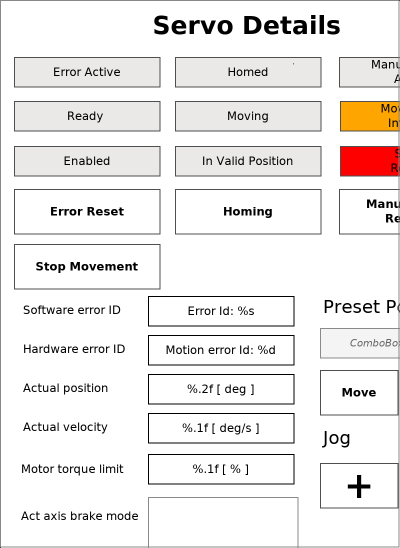
VISUALIZATION vAxisDetail  // 400x548
VAR_IN_OUT
	fbAxis: fb_ServoAxis;
	fbTableControl :FB_TableControl;
END_VAR
    Rectangle (0,0 495x856)
    Rectangle (339,189 146x45), "Manual mode Request", colour toggle: fbAxis.stHMI.bManualModeRequest
        toggle fbAxis.stHMI.bManualModeRequest
    Label (20,376 130x24), "Actual position"
    Label (20,415 130x24), "Actual velocity"
    Label (18,457 145x24), "Motor torque limit"
    Label (20,298 130x24), "Software error ID"
    Label (20,337 130x24), "Hardware error ID"
    Label (18,504 130x24), "Act axis brake mode"
    Label (18,544 130x24), "New brake mode"
    Frame (148,497 150x130)
        shows vAxisBrakeControl(fbData := MAIN.fbTableAxis)
    Rectangle (320,463 78x45), "+", colour toggle: fbAxis.stHMI.bJogForwardButton, input disabled if: fbAxis.iWorkStep_Axis<>15
        OnMouseDown: execute { fbAxis.stHMI.bJogForwardButton:=TRUE; }
        OnMouseLeave: execute { fbAxis.stHMI.bJogForwardButton :=FALSE; }
        OnMouseUp: execute { fbAxis.stHMI.bJogForwardButton :=FALSE; }
    Rectangle (405,463 74x45), "-", colour toggle: fbAxis.stHMI.bJogBackwardButton, input disabled if: fbAxis.iWorkStep_Axis<>15
        OnMouseDown: execute { fbAxis.stHMI.bJogBackwardButton:=TRUE; }
        OnMouseLeave: execute { fbAxis.stHMI.bJogBackwardButton:=FALSE; }
        OnMouseUp: execute { fbAxis.stHMI.bJogBackwardButton:=FALSE; }
    Label (149,8 196x34), "Servo Details"
    ComboBoxInteger (320,328 150x30), variable: fbAxis.stHMI.iManualPositionSelected, input disabled if: fbAxis.iWorkStep_Axis<>15
    Rectangle (320,370 78x45), "Move", colour toggle: fbAxis.stHMI.bGoToSelectedPosition, input disabled if: fbAxis.iWorkStep_Axis<>15
        OnMouseDown: execute { fbAxis.stHMI.bGoToSelectedPosition:=TRUE; }
        OnMouseLeave: execute { fbAxis.stHMI.bGoToSelectedPosition:=FALSE; }
        OnMouseUp: execute { fbAxis.stHMI.bGoToSelectedPosition:=FALSE; }
    Label (320,423 161x30), "Jog"
    Label (320,292 161x30), "Preset Position"
    Rectangle (175,189 146x45), "Homing", colour toggle: fbAxis.iWorkStep_Axis =20 OR fbAxis.iWorkStep_Axis =21
        OnMouseDown: execute { fbAxis.mFullHoming(); }
    Rectangle (339,57 146x30), "Manual mode Active", colour toggle: fbAxis.iWorkStep_Axis=15
    Rectangle (14,57 146x30), "Error Active", colour toggle: fbAxis.prIsErrorActive
    Rectangle (148,374 146x30), "%.2f [ deg ]", text variable: fbAxis.McReadActualPosition.Axis.NcToPlc.ModuloActPos
    Rectangle (148,413 146x30), "%.1f [ deg/s ]", text variable: fbAxis.McReadActualVelocity.ActualVelocity
    Rectangle (148,296 146x30), "Error Id: %s", text variable: TO_STRING(fbAxis.nActEvent)
    Rectangle (148,335 146x30), "Motion error Id: %d", text variable: fbAxis.udiActErrorCode
    Rectangle (148,454 146x30), "%.1f [ % ]", text variable: fbAxis.McTorqueMonitor.rTorqueLimit
        OnMouseClick: write the text variable via Default, min 1, max 100, title 'Motor torque limitation'
    Rectangle (175,57 146x30), "Homed", colour toggle: fbAxis.stHMI.bIsHomed
    Rectangle (14,101 146x30), "Ready", colour toggle: fbAxis.stHMI.bIsReady
    Rectangle (175,101 146x30), "Moving", colour toggle: fbAxis.stHMI.bIsMoving
    Rectangle (14,189 146x45), "Error Reset"
        OnMouseDown: execute { fbAxis.mErrorReset(); }
    Rectangle (340,101 146x30), "Movement Interlock", colour toggle: fbAxis.bMovementInterlock
    Rectangle (14,244 146x45), "Stop Movement"
        OnMouseDown: execute { fbAxis.stHMI.bRequestStopAxis:=TRUE; }
    Ellipse (293,63 0x1)
    Rectangle (14,146 146x30), "Enabled", colour toggle: fbAxis.prEnabled
    Rectangle (165,787 164x54), "CLOSE"
        OnMouseDown: execute { fbTableControl.stHMI.iDialogNumber:=0; }
    Rectangle (175,146 146x30), "In Valid Position", colour toggle: fbAxis.bPositionValid
    Rectangle (148,585 150x30), "%d [deg/s]", text variable: fbAxis.stSettings.rFastSpeed_deg_s
        OnMouseClick: write the text variable via Default, min 0, max 250, title 'Fast Speed', format %d
    Label (18,588 130x24), "Fast Speed"
    Rectangle (148,623 150x30), "%d [deg/s]", text variable: fbAxis.stSettings.rSlowSpeed_deg_s
        OnMouseClick: write the text variable via Default, min 0, max 100, title 'Slow Speed', format %d
    Label (18,626 130x24), "Slow Speed"
    Rectangle (148,663 150x30), "%d [deg/s2]", text variable: fbAxis.stSettings.rAcceleration
        OnMouseClick: write the text variable via Default, min 0, max 1000, title 'Acceleration', format %d
    Label (18,666 130x24), "Acceleration"
    Rectangle (148,701 150x30), "%d [deg/s2]", text variable: fbAxis.stSettings.rDeceleration
        OnMouseClick: write the text variable via Default, min 0, max 1000, title 'Deceleration', format %d
    Label (18,704 130x24), "Deceleration"
    Rectangle (148,740 150x30), "%d [deg]", text variable: fbAxis.stSettings.lrPositionTolerance
        OnMouseClick: write the text variable via Default, min 0, max 2, title 'Tolerance', format %.1f
    Label (18,741 130x24), "Position Tolerance"
    Rectangle (340,146 146x30), "Safety Release", colour toggle: fbAxis.bEnableMotion
    Checkbox (315,587 168x30), "Enable Quick Homing", variable: fbAxis.stSettings.bEN_QuickHoming
    Rectangle (315,663 150x30), "%.2f [deg]", text variable: fbAxis.lrReferencePositionAtHomeSensor
        OnMouseClick: write the text variable via Default, min 0, max 100, title 'Slow Speed', format %d
    Rectangle (315,740 150x30), "%.2f [deg]", text variable: fbAxis.lrLastPositionAtHomeSensor
        OnMouseClick: write the text variable via Default, min 0, max 100, title 'Slow Speed', format %d
    Label (315,705 130x24), "Last Home Position"
    Label (315,628 162x24), "Reference Home Position"
END_VISUALIZATION

(* stored: Version 1.1.0.1, ProductVersion 3.1.4024.15
   Visu vAxisDetail: Id {640b9dfd-7800-4663-98d3-1bae21fdd60e} *)
